{attribute addProperty BoxType "EP2001-1000-0016"}
{attribute addProperty Id "Output5AT %Q*BOOL811Output6AT %Q*BOOL812Output7AT %Q*BOOL813Output8AT %Q*BOOL814"}
{attribute addProperty CRC "2486434957"}
{attribute addProperty SizeInBites "32"}
{attribute addProperty SizeInBytes "4"}
TYPE Group_9433FC8D :
STRUCT
	{attribute addProperty Name "Output5"}
	Output5 AT %Q* : BOOL;
	{attribute addProperty Name "Output6"}
	Output6 AT %Q* : BOOL;
	{attribute addProperty Name "Output7"}
	Output7 AT %Q* : BOOL;
	{attribute addProperty Name "Output8"}
	Output8 AT %Q* : BOOL;
END_STRUCT
END_TYPE

(* stored: Version 1.2.0.0, ProductVersion 3.1.4024.9
   DUT Group_9433FC8D: Id {a5e8266b-f61d-4aac-90c6-953d310f747e} *)
